(*
SPDX-FileCopyrightText: © 2026 Oleksandr Tiutyk <trofimich@gmail.com>
SPDX-License-Identifier: MIT
License: https://opensource.org/license/mit
*)

(*!
<summary>Renames a file through cyclic task execution.</summary>
<description>
Use one owner task. Configure both paths, target, path type and timeout before Start and keep them unchanged
until STOPPED. Both paths are required during execution. The native service determines path and destination
collision behavior; this wrapper adds no overwrite, retry or rollback policy and reports native errors through
Task failure handling. Continue Execute through stopping after cancellation; pending native work must finish.
Failure or cancellation does not prove the original names were preserved. Reset preserves configuration.
</description>
*)

{attribute 'no_explicit_call' := 'do not call this function block directly'}
FUNCTION_BLOCK RenameFile EXTENDS TOF_Tasks.Task IMPLEMENTS IFileSystemTask
VAR_STAT
	//! <summary>Static type metadata available before the base task initializes its default name.</summary>
	{attribute 'hide'}
	_ClassName : STRING := __POUNAME();
END_VAR
VAR
    _RenameFile : Tc2_System.FB_FileRename;
END_VAR

(*!
<summary>Selects the ADS target for the native filesystem operation.</summary>
<description>
Configure before Start and keep unchanged until STOPPED; the setter stores configuration without submitting
I/O.
</description>
*)
{attribute 'monitoring' := 'call'}
{attribute 'OPC.UA.DA.Property' := '1'}
{attribute 'OPC.UA.DA' := '1'}
PROPERTY AmsNetId : Tc2_System.T_AmsNetID
GET
AmsNetId := _RenameFile.sNetId;
END_GET
SET
_RenameFile.sNetId := AmsNetId;
END_SET
END_PROPERTY

(*!
<summary>Provides the concrete type name used in diagnostics.</summary>
<description>
Returns borrowed read-only metadata; keep the instance alive and do not modify the referenced string.
Initialized static storage is ready during base Task.FB_init; this getter has no side effects or exceptions.
</description>
*)
{attribute 'monitoring' := 'call'}
PROPERTY ClassName : REFERENCE TO STRING
GET
ClassName REF= _ClassName;
END_GET
END_PROPERTY

(*!
<summary>Provides the library namespace used in diagnostics.</summary>
<description>Returns borrowed read-only namespace storage; do not modify the referenced string.</description>
*)
{attribute 'monitoring' := 'call'}
PROPERTY NamespaceName : REFERENCE TO STRING
GET
NamespaceName REF= CurrentNamespace.Name;
END_GET
END_PROPERTY

(*!
<summary>Provides the requested destination path for the rename operation.</summary>
<description>
Configure before Start and keep unchanged until STOPPED. Assignment does not reserve the destination or
guarantee replacement of an existing entry. Native collision behavior applies; Reset preserves it.
</description>
*)
{attribute 'monitoring' := 'call'}
{attribute 'OPC.UA.DA.Property' := '1'}
{attribute 'OPC.UA.DA' := '1'}
PROPERTY NewFilePath : Tc2_System.T_MaxString
GET
NewFilePath := _RenameFile.sNewName;
END_GET
SET
_RenameFile.sNewName := NewFilePath;
END_SET
END_PROPERTY

(*!
<summary>Provides the source path for the rename operation.</summary>
<description>
Configure before Start and keep unchanged until STOPPED. The setter copies text; native execution checks the
source. Reset preserves it.
</description>
*)
{attribute 'monitoring' := 'call'}
{attribute 'OPC.UA.DA.Property' := '1'}
{attribute 'OPC.UA.DA' := '1'}
PROPERTY OldFilePath : Tc2_System.T_MaxString
GET
OldFilePath := _RenameFile.sOldName;
END_GET
SET
_RenameFile.sOldName := OldFilePath;
END_SET
END_PROPERTY

(*!
<summary>Resets the native request edge after the task has stopped.</summary>
<description>
Preserves configured inputs and does not undo completed filesystem effects. Pending I/O must finish during
stopping before this hook runs.
</description>
*)
METHOD PROTECTED OnReset
_RenameFile(bExecute := FALSE);
END_METHOD

(*!
<summary>Submits and advances native renaming of the configured file.</summary>
<description>
Validates required configuration before submitting the request. Native errors raise an exception for the base
Task failure/stopping path without dynamic string-builder allocations. Normal completion reports DONE only
after the native block is no longer busy. No rollback is performed.
</description>
<param name="processingState">BUSY while pending; DONE after native completion without an error.</param>
<param name="stopReasonMessage">Not changed here; failures are passed through exceptions.</param>
*)
METHOD PROTECTED OnRunning
VAR_OUTPUT
	processingState : TOF_Tasks.TASK_PROCESSING_STATE;
END_VAR
VAR_IN_OUT
	stopReasonMessage : TOF_Core.ERROR_MESSAGE;
END_VAR
VAR
	formattedExceptionMessage : TOF_Core.ERROR_MESSAGE;
END_VAR
IF NOT _RenameFile.bExecute THEN 
	IF TOF_Core.Strings.IsNullOrWhiteSpace(stringToCheck := _RenameFile.sOldName) THEN
		TOF_Core.Exceptions.ThrowDataMemberNotSpecified(
			sourceNamespaceName := NamespaceName,
			sourceClassName := ClassName,
			sourcePOUName := __POUNAME(),
			sourcePosition := __POSITION(),
			dataMemberName := 'OldFilePath'
		);		
	END_IF

	IF TOF_Core.Strings.IsNullOrWhiteSpace(stringToCheck := _RenameFile.sNewName) THEN
		TOF_Core.Exceptions.ThrowDataMemberNotSpecified(
			sourceNamespaceName := NamespaceName,
			sourceClassName := ClassName,
			sourcePOUName := __POUNAME(),
			sourcePosition := __POSITION(),
			dataMemberName := 'NewFilePath'
		);		
	END_IF
	
	_RenameFile(bExecute := FALSE);
END_IF

_RenameFile(bExecute := TRUE);

IF _RenameFile.bError THEN
	TOF_Core.WideStrings.Append255(
		formattedExceptionMessage,
		"An error occurred while renaming the file '",
		TO_WSTRING(_RenameFile.sOldName),
		"' to '",
		TO_WSTRING(_RenameFile.sNewName),
		"'");

	FileSystemExceptions.ThrowFileSystem(
		sourceNamespaceName := NamespaceName,
		sourceClassName := ClassName,
		sourcePOUName := __POUNAME(),
		sourcePosition := __POSITION(),
		message := formattedExceptionMessage,
		errorCode := _RenameFile.nErrId
	);
END_IF

IF NOT _RenameFile.bBusy THEN
	processingState := TOF_Tasks.TASK_PROCESSING_STATE.DONE;
END_IF
END_METHOD

(*!
<summary>Waits for an already submitted operation before task termination.</summary>
<description>
Runs for every stop reason. Advances the pending FB with bExecute=FALSE without issuing another request.
Completion does not roll back side effects. Keep configuration and borrowed buffers valid until STOPPED.
</description>
<param name="readyToRelease">TRUE when the underlying FB is no longer busy.</param>
*)
METHOD PROTECTED OnStopping
VAR_OUTPUT
	readyToRelease : BOOL;
END_VAR
IF _RenameFile.bBusy THEN
	_RenameFile(bExecute := FALSE);
END_IF

readyToRelease := NOT _RenameFile.bBusy;
END_METHOD

(*!
<summary>Selects the native path context for the filesystem request.</summary>
<description>
Configure before Start and keep unchanged until STOPPED. It is passed to the native operation, not used as a
path-validity result. Reset preserves it.
</description>
*)
{attribute 'monitoring' := 'call'}
{attribute 'OPC.UA.DA.Property' := '1'}
{attribute 'OPC.UA.DA' := '1'}
PROPERTY PathType : Tc2_System.E_OpenPath
GET
PathType := _RenameFile.ePath;
END_GET
SET
_RenameFile.ePath := PathType;
END_SET
END_PROPERTY

(*!
<summary>Reports the size of this concrete instance in bytes.</summary>
*)
{attribute 'monitoring' := 'call'}
PROPERTY SelfSize : ULINT
GET
SelfSize := XSIZEOF(THIS^);
END_GET
END_PROPERTY

(*!
<summary>Configures the timeout passed to native operation requests.</summary>
<description>
Set before Start and keep unchanged until STOPPED. Reset preserves this value. It is not an overall task
deadline or a guarantee of resource release after a timeout.
</description>
*)
{attribute 'monitoring' := 'call'}
{attribute 'OPC.UA.DA.Property' := '1'}
{attribute 'OPC.UA.DA' := '1'}
PROPERTY Timeout : TIME
GET
Timeout := _RenameFile.tTimeout;
END_GET
SET
_RenameFile.tTimeout := Timeout;
END_SET
END_PROPERTY

END_FUNCTION_BLOCK

(* stored: Version 1.1.0.1
   POU RenameFile: Id {5fe3dd9c-88bf-4d47-ad86-126c81bbb806}, SpecialFunc None
   Folder Inputs: Id {64411f2c-4edc-4003-b87f-c74c67e7af3d}
   Folder Members to override: Id {55d19e21-d8e0-4806-9c88-3bb0901b741c}
   Property AmsNetId: Id {32a5c0ba-3c09-49c8-928e-dd03a2893039}
   Get Get: Id {bd483b3d-0ae6-43ac-bb9e-630766d488fd}
   Set Set: Id {1a7ac081-889f-4e41-8e19-e61735557134}
   Property ClassName: Id {f3928af8-0f1f-4879-92ca-79a10f3d7fe6}
   Get Get: Id {19cf5209-9aea-45f8-9d19-2a70acea8736}
   Property NamespaceName: Id {b0b906a0-5b5b-4052-8f97-2e660a46c7a9}
   Get Get: Id {2794b649-927b-49a0-84a1-b39c31e7029c}
   Property NewFilePath: Id {9cee3dbc-7338-4b33-bd95-a34d03b7caef}
   Get Get: Id {d64d0129-2bfe-4fa7-a8d2-7a545d94b5bb}
   Set Set: Id {09693386-a63b-476c-ac28-7df442f9f7df}
   Property OldFilePath: Id {8db36151-b36f-4fdb-aae6-f9fd8e6b59fd}
   Get Get: Id {9153f1f5-30bf-4c0c-a2fb-e6e367bbae32}
   Set Set: Id {d703ae33-46f0-4791-8d6d-83fda6da00a2}
   Method OnReset: Id {eb00bf66-c45d-4510-b44e-c13f9f91eb14}
   Method OnRunning: Id {2d8f899d-72fc-434c-81ad-005e64f50e2e}
   Method OnStopping: Id {55c27d00-9aad-474b-8b43-f6d5fe1f1f1c}
   Property PathType: Id {01c1abdf-1153-4312-b60e-df071bbd022a}
   Get Get: Id {c059cbff-ec88-4355-9f6d-596b0e46373e}
   Set Set: Id {46c2f573-ada2-4def-a399-dc1f5fcbb1bf}
   Property SelfSize: Id {88475cf2-6927-4fc3-9fcb-9b985365fa5f}
   Get Get: Id {43c07c8a-a1f8-4bba-a236-75e07e95cef8}
   Property Timeout: Id {170793eb-5a59-4f6b-ae58-a29f97e7fa7a}
   Get Get: Id {e9c2aeef-65a1-4409-93c1-4007b4099584}
   Set Set: Id {a16cebf2-d9ce-4fc3-8f0a-39d2c656bf15} *)
